// TwinCAT 3 PLC project main
// ProgramVersion: 3.1.4023.0
// libraries:
//   Tc2_Standard, * (Beckhoff Automation GmbH)
//   Tc2_System, * (Beckhoff Automation GmbH)
//   Tc3_Module, * (Beckhoff Automation GmbH)
// project tree:
//   DUTs/ State.TcDUT (not stored), StateSeparator.TcDUT
//   / PlcTask.TcTTO (not stored)
//   POUs/ FB_Separator.TcPOU (not stored), MAIN.TcPOU

// ---- DUTs/StateSeparator.TcDUT
{attribute 'qualified_only'}
{attribute 'strict'}
TYPE StateSeparator :
(
	Off,
	Init,
	Init_Wait,
	Ready,
	Eject,
	Eject_Wait_1,
	Eject_Wait_2,
	Done_Wait,
	Done
);
END_TYPE

// ---- POUs/MAIN.TcPOU
PROGRAM MAIN
VAR
	ModuleSeperationSensors 		AT%I*		: BYTE := 0;			// 0000_0dmu
	ModuleSeperationActuators		AT%Q*		: BYTE := 0;			// 0000_00rc
	
	sensUp, sensMiddle, sensDown				: BOOL;
	
	sigCreate, sigRemove				: BOOL;
	actUpOpen, actUpClose				: BOOL;
	actDownOpen, actDownClose 			: BOOL;
	
	moduleSeperation		: FB_Separator;
	seperationEnable, seperationExecute	: BOOL;
END_VAR

// Converting Inputs
sensUp := BYTE_TO_BOOL(ModuleSeperationSensors AND 2#0000_0001);
sensMiddle := BYTE_TO_BOOL(ModuleSeperationSensors AND 2#0000_0010);
sensDown := BYTE_TO_BOOL(ModuleSeperationSensors AND 2#0000_0100);


// Instance calls
moduleSeperation(
	bEnable:= seperationEnable, 
	bExecute:= seperationExecute, 
	bErrorReset:= , 
	bSensor1:= sensDown, 
	bSensor2:= sensMiddle, 
	bSensor3:= sensUp, 
	bR1AKT1=> actUpClose, 
	bR2AKT1=> actUpOpen, 
	bR1AKT2=> actDownOpen, 
	bR2AKT2=> actDownClose, 
	bNoBottle=> , bWrongBottle=> , eStatus=> );


// Converting Outputs
ModuleSeperationActuators := 0;
ModuleSeperationActuators := BOOL_TO_BYTE(sigCreate) OR ModuleSeperationActuators;
ModuleSeperationActuators := SHL(BOOL_TO_BYTE(sigRemove),1) OR ModuleSeperationActuators;

ModuleSeperationActuators := SHL(BOOL_TO_BYTE(actUpOpen),7) OR ModuleSeperationActuators;
ModuleSeperationActuators := SHL(BOOL_TO_BYTE(actUpClose),6) OR ModuleSeperationActuators;
ModuleSeperationActuators := SHL(BOOL_TO_BYTE(actDownOpen),5) OR ModuleSeperationActuators;
ModuleSeperationActuators := SHL(BOOL_TO_BYTE(actDownClose),4) OR ModuleSeperationActuators;

END_PROGRAM
